(* CoDeSys 2.3 export: MonitorReal.EXP *)

(* POU basic/MonitorReal, ST *)
FUNCTION MonitorReal : BOOL
VAR_INPUT
    Value: REAL;
    Channel: UINT;
END_VAR
VAR_IN_OUT
    Data: REAL;
END_VAR
VAR
END_VAR
IF Value <> Data THEN
    IF Channel < 256 THEN
        EvtCh8Tick32Real32(UINT_TO_BYTE(Channel), GlobalTick, Value, GlobalLogBufferHandle);
    ELSE
        EvtCh16Tick32Real32(Channel, GlobalTick, Value, GlobalLogBufferHandle);
    END_IF
    Data := Value;
END_IF
END_FUNCTION
